// TIA Portal V18 export
TYPE "UDT_Store_Setpoints"
// stored: IsFailsafeCompliant false
   STRUCT
      Room : Struct
         Actual : Struct
            rRATHeating : Real;
            rRATCooling : Real;
            rIAQ : Real;
            rBuildingdP : Real;
         END_STRUCT;
         Comfort : Struct
            rRATHeating : Real := 18.0;
            rRATCooling : Real := 22.0;
            rIAQ : Real := 600.0;
            rBuildingdP : Real := 5.0;
         END_STRUCT;
         PreComfort : Struct
            rRATHeating : Real := 16.0;
            rRATCooling : Real := 25.0;
            rIAQ : Real := 800.0;
            rBuildingdP : Real := 2.0;
         END_STRUCT;
         Econom : Struct
            rRATHeating : Real := 15.0;
            rRATCooling : Real := 30.0;
            rIAQ : Real;
            rBuildingdP : Real;
         END_STRUCT;
         Protection : Struct
            rRATHeating : Real := 5.0;
            rRATCooling : Real := 35.0;
            rIAQ : Real := 0.0;
            rBuildingdP : Real := 0.0;
         END_STRUCT;
      END_STRUCT;
   END_STRUCT;
END_TYPE
